Staubli VAL3: size_grid.pgx

program size_grid()
  local num l_nGridMax[2]
begin

  // helpers
  resize(nGrid,1,1)
  resize(nGrid,2,1)
  nGrid[0,0]=0

  // size grid
  call util:vecMax(nX1, l_nGridMax[0])
  call util:vecMax(nX2, l_nGridMax[1])
  resize(nGrid,1,max(l_nGridMax[0], l_nGridMax[1])+1)

  call util:vecMax(nY1, l_nGridMax[0])
  call util:vecMax(nY2, l_nGridMax[1])
  resize(nGrid,2,max(l_nGridMax[0], l_nGridMax[1])+1)
end
